// Mitsubishi GX Works2 project: MPS 장비 제어하기 1   PLC: Q03UDV

PROGRAM MAIN
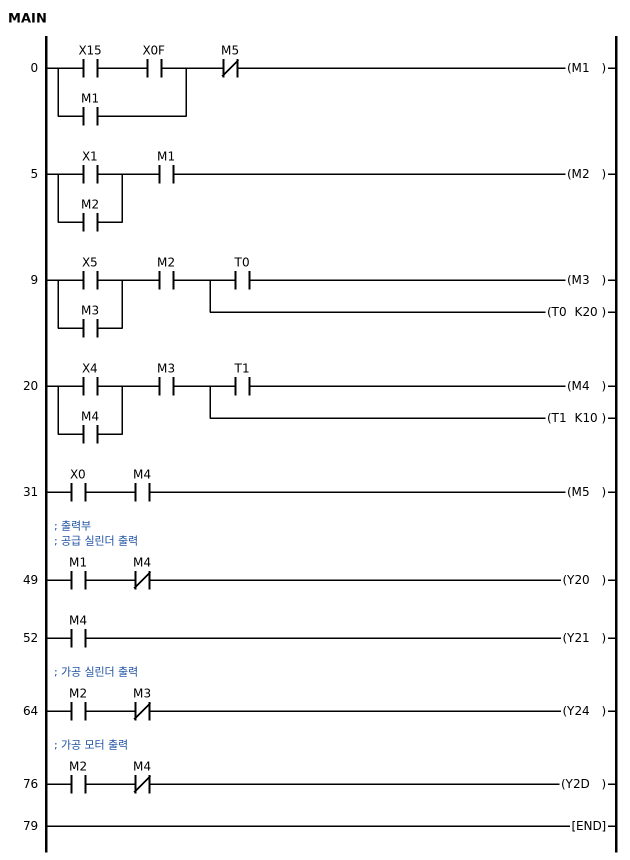
0     LD      X15
      AND     X0F
      OR      M1
      ANI     M5
      OUT     M1
5     LD      X1
      OR      M2
      AND     M1
      OUT     M2
9     LD      X5
      OR      M3
      AND     M2
      MPS
      AND     T0
      OUT     M3
      MPP
      OUT     T0 K20
20    LD      X4
      OR      M4
      AND     M3
      MPS
      AND     T1
      OUT     M4
      MPP
      OUT     T1 K10
31    LD      X0
      AND     M4
      OUT     M5
; 출력부
; 공급 실린더 출력
49    LD      M1
      ANI     M4
      OUT     Y20
52    LD      M4
      OUT     Y21
; 가공 실린더 출력
64    LD      M2
      ANI     M3
      OUT     Y24
; 가공 모터 출력
76    LD      M2
      ANI     M4
      OUT     Y2D
79    END
END_PROGRAM
